FUNCTION_BLOCK Ass_Sealing IMPLEMENTS ITF_AutoStructCommand
VAR_INPUT
END_VAR
VAR_OUTPUT
END_VAR
VAR
	i	:INT;
	_bProcessScan,_bInitialScan: BOOL;
	_bHalt , _bError,_bHaltPause: BOOL;
	strText	:STRING;
	nStep,nInitiStep ,nNextStep 	: INT;
	_tmrT0			:TON;
END_VAR

IF NOT _bInitialScan THEN
	nInitiStep	:= 0;
END_IF

_bInitialScan:=FALSE;



IF NOT _bProcessScan THEN
	nNextStep	:= 0;
	nStep		:= 0;
END_IF

_bProcessScan	:=FALSE;

PROPERTY Connect : STRING(50)
GET
CASE nStep OF
	5:
	Connect	:= 'OpenBox In';
	20:
	Connect	:= 'Ready'; 
	50:
	Connect	:= 'LoadPic In';
	ELSE	
	Connect	:= '';		
END_CASE
END_GET
SET
END_SET
END_PROPERTY

{warning 'add property implementation'}
PROPERTY Error : BOOL
GET
END_GET
END_PROPERTY

{warning 'add method implementation '}
METHOD ErrorClear : BOOL
END_METHOD

{warning 'add method implementation '}
METHOD FB_init : BOOL
VAR_INPUT
	(* if TRUE, the retain variables are initialized (warm start / cold start)*)
	bInitRetains	: BOOL;
	(* if TRUE, the instance afterwards gets moved into the copy code (online change)*)
	bInCopyCode	: BOOL;
END_VAR
END_METHOD

{warning 'add method implementation '}
METHOD HaltStepContiune : BOOL
END_METHOD

METHOD Initialization : BOOL
VAR_INPUT
	_Testmode	: BOOL;
END_VAR

VAR
	bConfig: BOOL;
END_VAR
_bInitialScan:=TRUE;

CASE nInitiStep OF
	0:		
		_tmrT0(IN:=FALSE);
		strText:='ORG : Initial ';
		Motor_BoxSealBottom_L.qRun		:=FALSE;
		Motor_BoxSealBottom_R.qRun		:=FALSE;
		Cyl_BeltBottomSup.qExtendCoil	:=FALSE;		
		nInitiStep						:= 5;
	5:
	bConfig			:=TRUE;
	IF Sen_BeltLoadIn OR Sen_BeltLoadOut THEN
		bConfig			:=FALSE;
		EventLogger.eEventType		:= 4;
		EventLogger.strEventText	:= 'Sensor Error ';	
		EventLogger();					
	END_IF		
	IF NOT Motor_BoxSealBottom_R.iError OR NOT Motor_BoxSealBottom_L.iError  THEN
		bConfig			:=FALSE;
		EventLogger.eEventType		:= 4;
		EventLogger.strEventText	:= 'INV. Motor Error ';	
		EventLogger();					
	END_IF	
	
	IF bConfig THEN
		strText:='ORG : Done ';
		nInitiStep	:= 20;
		ELSE
		strText:='ORG : Failed ';
		nInitiStep	:= 50;
	END_IF
	
	
	
	
	

20:
	Initialization	:= TRUE;

END_CASE;
END_METHOD

{warning 'add property implementation'}
PROPERTY NoEntry : BOOL
GET
END_GET
END_PROPERTY

{warning 'add method implementation '}
METHOD Pause : BOOL
END_METHOD

METHOD Process : BOOL
VAR_INPUT
	bHlatMode	: BOOL;
END_VAR


_bProcessScan	:= TRUE;
//判斷 

IF _bError THEN
	strText	:= 'OpenBox:Error ';
	strText	:= CONCAT(Status,INT_TO_STRING(nStep));
END_IF;
//半自動模式
IF NOT bHlatMode  THEN
	nStep:= nNextStep;	
END_IF;

_bHaltPause	:= nStep<> nNextStep;
IF _bError OR _bHaltPause THEN
	RETURN;
END_IF

//主程序 
IF NOT _bHaltPause THEN
	CASE nStep OF
		0:
			_tmrT0(IN:=FALSE);
			Motor_BoxSealBottom_L.qRun		:=TRUE;
			Motor_BoxSealBottom_R.qRun		:=TRUE;
			nNextStep						:= 5;
			strText							:= 'Waiting for load';
		5:
			IF Sen_BeltLoadIn THEN
				Cyl_BeltBottomSup.qExtendCoil	:=TRUE;
				strText							:= 'load In';
				nNextStep						:= 10;
			END_IF;	
		10:
			IF NOT Sen_BeltLoadIn THEN
				//Cyl_BeltBottomSup.qExtendCoil	:=FALSE;
				;
			END_IF;		
	
			IF Sen_BeltLoadOut THEN
				Cyl_BeltBottomSup.qExtendCoil	:=FALSE;
				strText						:= 'load Out';
				nNextStep					:= 15;
			END_IF;		
		15:
			_tmrT0(IN:=TRUE,PT:=T#0.5S);
			IF _tmrT0.Q THEN
				_tmrT0(IN:=FALSE);
				IF OP.xAutoMode THEN
					nNextStep					:= 20;
					ELSE
					nNextStep					:= 50;
				END_IF;
			END_IF
		20:
				IF M_LoadPic3.Connect= 'Seal In' THEN
					nNextStep					:= 21;
					ELSE
					Motor_BoxSealBottom_L.qRun		:=FALSE;
					Motor_BoxSealBottom_R.qRun		:=FALSE;
				END_IF
		21:
				_tmrT0(IN:=NOT Sen_BeltLoadOut,PT:=T#0.5S);
				Motor_BoxSealBottom_L.qRun		:=TRUE;
				Motor_BoxSealBottom_R.qRun		:=TRUE;		
				IF 	_tmrT0.Q THEN
					_tmrT0(IN:=FALSE);
					nNextStep					:= 50;
				END_IF
		50:
				nNextStep					:= 0;
	END_CASE
END_IF;

Process	:= nStep =50;
END_METHOD

{warning 'add property implementation'}
PROPERTY Status : STRING(50)
GET
END_GET
END_PROPERTY

END_FUNCTION_BLOCK

(* stored: Version 1.1.0.1, ProductVersion 3.1.4026.18
   POU Ass_Sealing: Id {25f63225-dbc9-4b1e-b86a-0e068b049cd3}, SpecialFunc None
   Property Connect: Id {83bd3ff5-c6e3-4a8c-8bba-d49023e80782}
   Get Get: Id {5d7475ec-f8cf-40fd-aa0d-db8e368e47ed}
   Set Set: Id {927d6ae5-1a73-4a7f-9841-6b22e665c0dd}
   Property Error: Id {c4e7731e-732d-489c-9847-7d733a800e09}
   Get Get: Id {ef07e930-46de-449d-b1ba-f8123ef084cf}
   Method ErrorClear: Id {4351c64a-5973-412f-9c2a-d62ab6ea446f}
   Method FB_init: Id {49c9e524-43f7-4b09-8037-50637c554f51}
   Method HaltStepContiune: Id {e067c393-fc75-436b-a825-48fad1a93c84}
   Method Initialization: Id {c0f7d7e1-8a43-4b52-b274-e8f58634f2e0}
   Property NoEntry: Id {7f044b28-0411-4954-86f6-f74c7f97a387}
   Get Get: Id {805ef038-e4f3-4be4-8390-1e1ba28c3bb3}
   Method Pause: Id {3248126b-b242-4316-ae47-c6ac4ef43604}
   Method Process: Id {bf7874d8-aa7d-4a83-9850-3952fbf34226}
   Property Status: Id {3522a825-d2b8-46c3-9396-824ffc70819e}
   Get Get: Id {ddbe10c8-e747-4091-b45b-68c48cded3b1} *)
